INTERFACE IInputDevice EXTENDS IDevice

METHOD ReadInputs
END_METHOD

END_INTERFACE

(* stored: Version 1.1.0.1
   Itf IInputDevice: Id {ee96199e-8788-4fb6-b050-ed776ced9cc6}
   Method ReadInputs: Id {9943c009-39d2-4860-b10a-f331d4106b45} *)
